// TIA Portal V20 export
// export: Created 2025-12-01T14:57:43.4316475Z, ExportSetting None, DisplayName Totally Integrated Automation Portal, DisplayVersion V20 Update 3, DisplayName TIA Portal Openness, DisplayVersion V20 Update 3, DisplayName TIA Portal Version Control Interface, DisplayVersion V20 Update 3, DisplayName STEP 7 Professional, DisplayVersion V20 Update 3, DisplayName STEP 7 Safety, DisplayVersion V20 Update 2, DisplayName WinCC Basic/Comfort/Advanced, DisplayVersion V20 Update 3, DisplayName WinCC Professional, DisplayVersion V20 Update 3, DisplayName WinCC Unified, DisplayVersion V20 Update 3
FUNCTION "FC502_Actualiza_FIFO_SCR" : Void   // FC502, LAD
{ S7_Optimized_Access := 'FALSE' }
AUTHOR : TLigero
NAME : 20180425
VERSION : 3.1
// stored: AutoNumber false, SetENOAutomatically false
   VAR_INPUT
      DB_FIFO_Ordenes : UInt;
      Num_Scanner : UInt;   // Numero de scanner sobre el que se realiza la busqueda
      Long_FIFO : UInt;
   END_VAR
   VAR_IN_OUT
      FIFO_OK : Bool;
   END_VAR
   VAR_TEMP
      relleno : Byte;
      Indice : Int;
      final : Int;
      retval : Int;
      posicion_actual_N : UInt;
      posicion_siguiente_N1 : UInt;
      Dato_fifo : "ROUT_Orden_Fifo_Scanner";
      Registro_Fifo_vacio : "ROUT_Orden_Fifo_Scanner";
   END_VAR
BEGIN

REGION Network 1 (SCL)
   REGION INICIALIZACIÓN

       #FIFO_OK := FALSE;
       #relleno := 0;
       #retval:= FILL(BVAL := #relleno, BLK => #Registro_Fifo_vacio);
       #posicion_actual_N := 1;
       #final := #Long_FIFO;

   END_REGION
END_REGION

REGION Network 2 (SCL)
   REGION FIFO_1_POS
       //si la fifo es de una posición con borrar esta ya es suficiente.

       IF #Long_FIFO = 1 THEN
           "FC572_Guardar_Datos_Fifo"(DB_FIFO_Ordenes := #DB_FIFO_Ordenes,
                                      Num_Scanner := #Num_Scanner,
                                      Long_FIFO := #Long_FIFO,
                                      Posicion_FIFO := #posicion_actual_N,
                                      Datos_Scanner_Cruce := #Registro_Fifo_vacio);

           #FIFO_OK := true;
           RETURN;

       END_IF;


   END_REGION
END_REGION

REGION Network 3 (SCL)
   REGION FIFO_VARIAS_POSICIONES

       FOR #Indice := 2 TO #final BY 1 DO
           "FC571_Leer_Datos_Fifo"(DB_FIFO_Ordenes:=#DB_FIFO_Ordenes,
                                   Num_Scanner:=#Num_Scanner,
                                   Long_FIFO:=#Long_FIFO,
                                   Posicion_FIFO:=#Indice,
                                   Datos_Scanner_Cruce=>#Dato_fifo);

           "FC572_Guardar_Datos_Fifo"(DB_FIFO_Ordenes:=#DB_FIFO_Ordenes,
                                      Num_Scanner:=#Num_Scanner,
                                      Long_FIFO:=#Long_FIFO,
                                      Posicion_FIFO:=(#Indice-1),
                                      Datos_Scanner_Cruce:=#Dato_fifo);

           "FC572_Guardar_Datos_Fifo"(DB_FIFO_Ordenes := #DB_FIFO_Ordenes,
                                      Num_Scanner := #Num_Scanner,
                                      Long_FIFO := #Long_FIFO,
                                      Posicion_FIFO := #Indice,
                                      Datos_Scanner_Cruce := #Registro_Fifo_vacio);

       END_FOR;
       #FIFO_OK := true;

   END_REGION
END_REGION
END_FUNCTION
